// TIA Portal V16 export
// export: Created 2021-07-03T21:22:41.6233336Z, ExportSetting WithDefaults, DisplayName Totally Integrated Automation Portal, DisplayVersion V16, DisplayName TIA Portal Version Control Interface, DisplayVersion V16, DisplayName TIA Portal Openness, DisplayVersion V16, DisplayName STEP 7 Professional, DisplayVersion V16, DisplayName STEP 7 Safety, DisplayVersion V16, DisplayName WinCC Professional, DisplayVersion V16
DATA_BLOCK "TRCV_C_DB"   // DB2
// stored: AutoNumber true, DBAccessibleFromOPCUA true, InstanceOfName TRCV_C, OfSystemLibElement TRCV_C, OfSystemLibVersion 3.2
"TRCV_C"
   // VAR_INPUT
   //    EN_R : Bool;
   //    CONT : Bool;
   //    LEN : UDInt;
   //    ADHOC : Bool;
   // END_VAR
   // VAR_OUTPUT
   //    DONE : Bool;
   //    BUSY : Bool;
   //    ERROR : Bool;
   //    STATUS : Word;
   //    RCVD_LEN : UDInt;
   // END_VAR
   // VAR_IN_OUT
   //    CONNECT : Variant;
   //    DATA : Variant;
   //    ADDR : Variant;
   //    COM_RST : Bool;
   // END_VAR
   // VAR
   //    s_state : Int;
   //    s_locked : Bool;
   //    s_udp : Bool;
   //    s_configured : Bool;
   //    s_tcon_80A3 : Bool;
   //    s_ConID : CONN_OUC;
   //    s_TCON { S7_SetPoint := 'True'} : TCON;
   //    s_TDIAG { S7_SetPoint := 'True'} : T_DIAG;
   //    s_TDIAG_Status { S7_SetPoint := 'True'} : TDiag_Status;
   //    s_TRCV { S7_SetPoint := 'True'} : TRCV;
   //    s_TURCV { S7_SetPoint := 'True'} : TURCV;
   //    s_TDISCON { S7_SetPoint := 'True'} : TDISCON;
   //    s_TRESET { S7_SetPoint := 'True'} : T_RESET;
   // END_VAR
BEGIN
END_DATA_BLOCK
